FUNCTION_BLOCK FB_SmartKeypad
VAR_INPUT
END_VAR
VAR_OUTPUT
END_VAR
VAR
END_VAR

END_FUNCTION_BLOCK

(* stored: Version 1.1.0.1, ProductVersion 3.1.4024.12
   POU FB_SmartKeypad: Id {17aeb602-d27e-4e0c-ac87-0edb14e64c01}, SpecialFunc None *)
